TYPE LREAL100FIFOBuffer :
STRUCT
	Size: UDINT := 100;
	Buffer: ARRAY [0..99] OF LREAL;
END_STRUCT
END_TYPE

(* stored: Version 1.1.0.1, ProductVersion 3.1.4024.9
   DUT LREAL100FIFOBuffer: Id {aa95bb0f-6b65-40bb-aa15-b7039915cbf0} *)
